FUNCTION InfluxAddData_1Hz : BOOL
VAR_IN_OUT
	Data			: ST_DATA;
	DataCollector	: FB_InfluxDataCollector;
END_VAR

// Damage counter values
DataCollector.AddLreal('Test2',		Data.Gps.Inputs.x);

END_FUNCTION

(* stored: Version 1.1.0.1, ProductVersion 3.1.4022.11
   POU InfluxAddData_1Hz: Id {8ffdae7d-952a-4dde-b564-0025ab744451}, SpecialFunc None *)
